(* CODESYS project KruisingSimpleV3Demo.project

Project tree, tasks and I/O mapping:
  CODESYS_Control_Win_V3 : CODESYS Control Win V3, 3S - Smart Software Solutions GmbH, version 3.5.13.20
    application Application
      libraries: Standard, 3.5.14.0 (System)
      task Task (cyclic, interval t#20ms, priority 1) calls Kruising_prg
  libraries: VisuSymbols, 3.5.10.0 (System); Standard64, * (System); Util, * (System); Standard, * (System)
  function block Verkeerslicht [ST]: gaGroen, isRood, GroenTijd, Cycle, Init
  data type LichtToestand
  program Kruising_prg [ST]
  text list GlobalTextList
*)

// LichtToestand
TYPE LichtToestand :
(
	Rood, Geel, Groen, GroenVerlopen
);
END_TYPE

// Kruising_prg
PROGRAM Kruising_prg
VAR
	fbVerkeerslichtA			: Verkeerslicht;
	fbVerkeerslichtB			: Verkeerslicht;
	xInitialized				: BOOL := FALSE;
	xToggle						: BOOL := FALSE;
END_VAR

fbVerkeerslichtA.Cycle();
fbVerkeerslichtB.Cycle();

IF NOT xInitialized THEN
	fbVerkeerslichtA.Init();
	fbVerkeerslichtB.Init();
	xInitialized := TRUE;
END_IF

IF fbVerkeerslichtA.isRood() AND NOT xToggle THEN
	fbVerkeerslichtB.gaGroen();
	xToggle := TRUE;
END_IF;

IF fbVerkeerslichtB.isRood() AND xToggle THEN
	fbVerkeerslichtA.gaGroen();
	xToggle := FALSE;
END_IF;

END_PROGRAM

// Verkeerslicht
FUNCTION_BLOCK Verkeerslicht
VAR
	xRoodAan		: BOOL;
	xGeelAan		: BOOL;
	xGroenAan		: BOOL;
	eToestand		: LichtToestand := Rood;
	xRoodGevraagd 	: BOOL;
	tGroenTijd		: TIME := T#10S;
	tGeelTijd		: TIME := T#3S;
	tonGroenTimer 	: TON;
	tonGeelTimer 	: TON;
END_VAR

// Constructor

// cycle through aggregated objects
tonGroenTimer(IN:=(eToestand=Groen),PT:=tGroenTijd);
tonGeelTimer(IN:=(eToestand=Geel),PT:=tGeelTijd);

CASE eToestand OF
Rood: // call event handled in goGreen()
Groen:
	IF tonGroenTimer.Q THEN
		xGroenAan := FALSE;
		eToestand := Geel;//GroenVerlopen;
		xGeelAan := TRUE;
	END_IF
GroenVerlopen: // call event handled in goRed()		
	IF xRoodGevraagd THEN
		xGroenAan := FALSE;				
		xRoodGevraagd := FALSE;		
		eToestand := Geel;
		xGeelAan := TRUE;
	END_IF
Geel:
	IF tonGeelTimer.Q THEN
		xGeelAan := FALSE;
		eToestand := Rood;
		xRoodAan := TRUE;		
	END_IF
END_CASE

METHOD PUBLIC gaGroen
VAR_INPUT
END_VAR
CASE eToestand OF
Rood:
	xRoodAan := FALSE;
	eToestand := Groen;
	xGroenAan := TRUE;	
END_CASE
END_METHOD

METHOD PUBLIC isRood : BOOL
VAR_INPUT
END_VAR
isRood := THIS^.xRoodAan;
END_METHOD

PROPERTY GroenTijd : TIME
SET
VAR
	tTijd: 	TIME;
END_VAR
tGroenTijd := tTijd;
END_SET
GET
	GroenTijd := tGroenTijd;
END_GET
END_PROPERTY

METHOD Cycle
VAR_INPUT
END_VAR
THIS^();
END_METHOD

METHOD PUBLIC Init
VAR_INPUT
END_VAR
// initialize attributes
eToestand := Rood;
xRoodAan := TRUE;

// initialize aggregated objects
   // No aggregated objects
END_METHOD

END_FUNCTION_BLOCK
